INTERFACE I_SessionIdGenerator

METHOD PUBLIC Generate : T_MAXSTRING
VAR_INPUT
END_VAR
END_METHOD

END_INTERFACE

(* stored: Version 1.1.0.1, ProductVersion 3.1.4026.13
   Itf I_SessionIdGenerator: Id {3a351f19-b827-4fd9-b989-5b6e918d8d70}
   Method Generate: Id {22f12bc9-ae6d-4229-b401-8cab5f2fb29a} *)
